(* CoDeSys 2.3 library: TcPlcUtilitiesBC.lb6 *)
(* Libraries: standard.lb6 5.6.98 11:03:02, PlcSystemBC.lb6 21.3.01 11:03:02 *)

(* Global variable list: Global_Variables *)
VAR_GLOBAL
	GLOBAL_DCF77_PULSE_SPLIT		: TIME := T#140ms;(* 0 == pulse < 140ms, 1 == pulse > 140 *)
	GLOBAL_DCF77_SEQUENCE_CHECK	: BOOL := FALSE;(* TRUE = Enable plausibility check (two telegrams are checked), FALSE = Disable check *)
END_VAR

(* Data type *)
TYPE E_ArgType :(

	ARGTYPE_UNKNOWN			:= 0,
	ARGTYPE_BYTE,
	ARGTYPE_WORD,
	ARGTYPE_DWORD,
	ARGTYPE_REAL,
	ARGTYPE_LREAL,
	ARGTYPE_SINT,
	ARGTYPE_INT,
	ARGTYPE_DINT,
	ARGTYPE_USINT,
	ARGTYPE_UINT,
	ARGTYPE_UDINT,
	ARGTYPE_STRING,
	ARGTYPE_TIME
);
END_TYPE

(* Data type *)
TYPE E_TimeZoneID :
(
	eTimeZoneID_Invalid 	:= -1,
	eTimeZoneID_Unknown  	:= 0,
	eTimeZoneID_Standard	:= 1,(* Winterzeit *)
	eTimeZoneID_Daylight 	:= 2(* Sommerzeit *)
);
END_TYPE

(* Data type *)
TYPE OTSTRUCT:
STRUCT
	wWeek:			WORD;
 	wDay:			WORD;
 	wHour:			WORD;
 	wMinute:			WORD;
 	wSecond:		WORD;
 	wMilliseconds:	WORD;
END_STRUCT
END_TYPE

(* Data type *)
TYPE T_Arg :
STRUCT
	eType				: E_ArgType			:= ARGTYPE_UNKNOWN;	(* Argument data type *)
	cbLen				: UDINT 				:= 0;							(* Argument data byte length *)
	pData				: UDINT 				:= 0;							(* Pointer to argument data *)
END_STRUCT
END_TYPE

(* Data type *)
TYPE TIMESTRUCT
STRUCT
	wYear			: WORD;
     	wMonth			: WORD;
     	wDayOfWeek		: WORD;
     	wDay			: WORD;
     	wHour			: WORD;
     	wMinute			: WORD;
     	wSecond		: WORD;
     	wMilliseconds 	: WORD;
END_STRUCT
END_TYPE

(* POU CLEARBIT32, ST *)
FUNCTION CLEARBIT32 : DWORD
VAR_INPUT
	inVal32	:	DWORD;
	bitNo	:	SINT;
END_VAR
VAR
	dwConst : DWORD := 1;
END_VAR
CLEARBIT32 := inVal32 AND NOT (SHL(dwConst,bitNo MOD 32));
END_FUNCTION

(* POU CSETBIT32, ST *)
FUNCTION CSETBIT32 : DWORD	(* conditional set bit in dword *)
VAR_INPUT
	inVal32	:	DWORD;
	bitNo	:	SINT;
	bitVal	:	BOOL;		(* value to which the bit should be set *)
END_VAR
VAR
	dwConst : DWORD := 1;
END_VAR
IF bitVal
THEN
	CSETBIT32 := inVal32 OR SHL(dwConst,bitNo MOD 32);
ELSE
	CSETBIT32 := inVal32 AND NOT (SHL(dwConst,bitNo MOD 32));
END_IF;
END_FUNCTION

(* POU DCF77_TIME, ST *)
FUNCTION_BLOCK DCF77_TIME
(* DCF77 decoder function block *)
VAR_INPUT
	DCF_PULSE	:BOOL; (* DCF77 pulse: 101010101... *)
	RUN		:BOOL; (* Enable/disable function block execution. *)
END_VAR
VAR_OUTPUT
	BUSY		:BOOL;(* TRUE = Decoding in progress *)
	ERR		:BOOL;(* Error flag: TRUE = Error, FALSE = No error *)
	ERRID		:UDINT;(* Error code *)
	ERRCNT	:UDINT;(* Error counter *)
	READY		:BOOL;  (* TRUE => CDT is valid, FALSE => CDT is not valid *)
	CDT		:DATE_AND_TIME;(* date and time information *)
END_VAR
(* 	Error codes:
	0x100	:Timeout error (no DCF-Signal)
	0x200	:Parity error
	0x300	:Wrong time or date values (e.g. Month=13)
	0x400	:Data cycle to long
	0x500	:Data cycle to short 
*)
VAR
	DataBits		: ARRAY[0..60] OF BOOL;
	BitNo		: BYTE;
	dtCurr		: DATE_AND_TIME;
	dtNext		: DATE_AND_TIME;
	tziCurr		: E_TimeZoneID;(* Time zone information extracted from latest telegram *)
	tziPrev		: E_TimeZoneID;(* Time zone information extracted from previous telegram *)
	tDiff			: TIME;(* Two telegram time difference *)
	bCheck		: BOOL := FALSE;
{library private}

	Step		: BYTE;
	StartEdge	: R_TRIG;

	RisingPulse	: R_TRIG;
	FallingPulse	: F_TRIG;
	LongPulse	: TON;
	ShortPulse	: TON;
	DetectSync	: TOF;
	NoDCFSignal	: TON;
	DCFCycleLen	: TON;

	bIsRising	: BOOL;
	bIsFalling	: BOOL;
	bIsLong		: BOOL;
	bIsShort		: BOOL;
	Working		: BOOL;

	DataValid	: BOOL;
	ParitySum1	: BYTE;
	ParitySum2	: BYTE;
	ParitySum3	: BYTE;

	i			: BYTE;
	DummyByte	: BYTE;
	DummyString	: STRING;

	Hour		: BYTE;
	Minute		: BYTE;
	Year		: BYTE;
	Month		: BYTE;
	Day			: BYTE;
{library public}
END_VAR
StartEdge( CLK := RUN );
IF  StartEdge.Q THEN
	bCheck			:= FALSE;
	BUSY			:= TRUE;
	ERR			:= FALSE;
	ERRID			:= 0;
	ERRCNT		:= 0;
	DataValid		:= FALSE;
	Working 			:= FALSE;
	BitNo			:= 0;
	NoDCFSignal( IN := FALSE );
	DCFCycleLen( IN := FALSE );
	DetectSync( IN := TRUE );
	RisingPulse( CLK := FALSE );
	FallingPulse( CLK := FALSE );
	Step			:= 10;	(* start decoding, wait for sync *)
ELSIF NOT RUN THEN
	BUSY			:= FALSE;
END_IF


IF BUSY THEN

	READY			:=FALSE;(*Ready=true is set only for one cycle*)

	RisingPulse( CLK:=DCF_PULSE ); (* detect rising edge *)
	bIsRising := RisingPulse.Q;
	FallingPulse( CLK:=DCF_PULSE );	(* detect falling edge *)
	bIsFalling := FallingPulse.Q;
	LongPulse( IN := DCF_PULSE, PT := GLOBAL_DCF77_PULSE_SPLIT );(* configurable split point *)
	IF LongPulse.Q THEN
		bIsLong := TRUE;
	END_IF
	ShortPulse( IN := DCF_PULSE, PT := T#30ms );
	IF ShortPulse.Q THEN
		bIsShort := TRUE;
	END_IF

	DetectSync( IN := DCF_PULSE, PT := T#1s500ms );(*detect the sync second*)
	IF NOT DetectSync.Q THEN
		BitNo 		:= 0;
		Step 		:= 20; (* wait for high *)
	END_IF


	NoDCFSignal( IN := DetectSync.Q, PT := T#2m );
	IF NoDCFSignal.Q THEN
		NoDCFSignal( IN := FALSE );
		ERRID		:=16#100;
		Step		:= 100;
	END_IF

	(*checking if the data cycle was longer as needed*)
	DCFCycleLen( IN:= Working , PT:=T#59s );
	IF DCFCycleLen.Q THEN
		DCFCycleLen( IN := FALSE );
		ERRID		:= 16#400;
		Step 		:= 100;
	END_IF

	CASE Step OF
		10:	(* start decoding, wait for sync *)
			BitNo := 0;

		20: (* wait for rising edge *)
			IF bIsRising THEN
				IF DataValid THEN
					DataValid 	:= FALSE;
					ERR 		:= FALSE;
					ERRID 		:= 0;
					ERRCNT 	:= 0;
					READY 		:= TRUE;
				END_IF

				IF BitNo = 0 THEN
					Working 	:= TRUE; (* set flag *)
				END_IF
				bIsLong 	:= FALSE;
				bIsShort 	:= FALSE;
				Step 		:= 30;  (* wait for falling edge *)
			END_IF

		30:	(* wait for falling pulses *)
			IF bIsFalling THEN
				IF bIsLong THEN (* long pulse *)
					DataBits[BitNo] := TRUE;
					BitNo:=BitNo+1;
				ELSIF bIsShort THEN (* short pulse *)
					DataBits[BitNo] := FALSE;
					BitNo:=BitNo+1;
				END_IF

				bIsShort := FALSE;
				bIsLong := FALSE;

				IF BitNo < 59 THEN
					Step := 20;	(* repeat *)
				ELSIF BitNo = 59 THEN
					(********************************************************************************************************)
					(*check the parity Bits....*)
					ParitySum1:=0;
					ParitySum2:=0;
					ParitySum3:=0;
					FOR i:=21 TO 28 DO (*add parity bits*)
						IF DataBits[i] THEN
							ParitySum1:=ParitySum1+1;
						END_IF
					END_FOR
					FOR i:=29 TO 35 DO
						IF DataBits[i] THEN
							ParitySum2:=ParitySum2+1;
						END_IF
					END_FOR
					FOR i:=36 TO 58 DO
						IF DataBits[i] THEN
							ParitySum3:=ParitySum3+1;
						END_IF
					END_FOR

					(*if no parity errors decode the data and set the time and date variables*)
					IF( ( ParitySum1 MOD 2 ) = 0 )
					AND ( ( ParitySum2 MOD 2 ) = 0 )
					AND ( ( ParitySum3 MOD 2 ) = 0 )
					AND ( DataBits[20] = 1 )
					AND ( DataBits[0] = 0 )
					THEN

						DummyByte:=0;
						FOR i:=21 TO 27 DO
							IF DataBits[ i ] THEN
								DummyByte := DummyByte OR SHL(BYTE#1, i - 21 );
							END_IF
						END_FOR
						Minute:= ( DummyByte AND 2#00001111 ) + ( SHR( DummyByte, 4 ) * 10 );

						DummyByte:=0;
						FOR i:=29 TO 34 DO
							IF DataBits[ i ] THEN
								DummyByte := DummyByte OR SHL(BYTE#1, i - 29 );
							END_IF
						END_FOR
						Hour:= ( DummyByte AND 2#00001111 ) + ( SHR( DummyByte, 4 ) * 10 );

						DummyByte:=0;
						FOR i:=36 TO 41 DO
							IF DataBits[ i ] THEN
								DummyByte := DummyByte OR SHL(BYTE#1, i - 36 );
							END_IF
						END_FOR
						Day := ( DummyByte AND 2#00001111 ) + ( SHR( DummyByte, 4 ) * 10 );

						DummyByte:=0;
						FOR i:=45 TO 49 DO
							IF DataBits[ i ] THEN
								DummyByte := DummyByte OR SHL(BYTE#1, i - 45 );
							END_IF
						END_FOR
						Month := ( DummyByte AND 2#00001111 ) + ( SHR( DummyByte, 4 ) * 10 );

						DummyByte:=0;
						FOR i:=50 TO 57 DO
							IF DataBits[ i ] THEN
								DummyByte := DummyByte OR SHL(BYTE#1, i - 50 );
							END_IF
						END_FOR
						Year := ( DummyByte AND 2#00001111 ) + ( SHR( DummyByte, 4 ) * 10 );

						(*Create date and time strings*)
						(*Year 2000 problem...*)
						DummyString:='DT#2';
						IF Year < 100 THEN
							DummyString:=CONCAT( DummyString, '0'  );
						END_IF
						IF Year < 10 THEN
							DummyString:=CONCAT( DummyString, '0'  );
						END_IF

						DummyString:=CONCAT( DummyString, BYTE_TO_STRING( Year ) );
						DummyString:=CONCAT( DummyString, '-'  );
						DummyString:=CONCAT( DummyString, BYTE_TO_STRING( Month ) );
						DummyString:=CONCAT( DummyString, '-' );
						DummyString:=CONCAT( DummyString, BYTE_TO_STRING( Day ) );
						DummyString:=CONCAT( DummyString, '-' );
						DummyString:=CONCAT( DummyString, BYTE_TO_STRING( Hour ) );
						DummyString:=CONCAT( DummyString, ':'  );
						DummyString:=CONCAT( DummyString, BYTE_TO_STRING( Minute ) );
						DummyString:=CONCAT( DummyString, ':00' );

						IF ( Minute > 59 ) OR ( Hour > 23 ) OR ( Day > 31 ) OR ( Day = 0 ) OR ( Month > 12 ) OR ( Month = 0 ) THEN
							ERRID		:= 16#300; (*invalid Values*)
							Step		:= 100;
						ELSE
							(*checking if the data cycle was shorter as needed*)
							IF ( DCFCycleLen.ET <T#58s ) THEN
								ERRID		:= 16#500;
								Step		:= 100;
							ELSE

								IF NOT ( DataBits[17] XOR DataBits[18] ) THEN(* bit17 = 0 and bit18 = 1 => MEZ (Standard, Winterzeit), bit17 = 1 and bit 18 = 0 => MESZ (Daylight, Sommerzeit) *)
									ERRID	:= 16#300; (*invalid MEZ/MESZ bit values*)
									Step	:= 100;
								ELSE

									dtCurr := STRING_TO_DT(DummyString);(* convert string to next time *)
	
									IF NOT GLOBAL_DCF77_SEQUENCE_CHECK THEN(* Old code: no telegram check *)
	
										DataValid	:= TRUE;
										Working		:= FALSE;
										CDT		:= dtCurr;
										BitNo 		:= 0;
										Step		:= 10;
	
									ELSE(* New code: check two telegrams *)

										IF bCheck THEN(* check the prev and current telegram*)
											tDiff := SEL( dtCurr > dtNext, dtNext - dtCurr, dtCurr - dtNext );
											tziCurr := SEL( DataBits[17], eTimeZoneID_Standard, eTimeZoneID_Daylight );

											IF ( dtNext = dtCurr )
											OR ( ( tDiff = T#1h )  AND ( tziCurr <> tziPrev ) AND DataBits[16] )(* MEZ->MESZ or MESZ->MEZ change *)
											THEN(* Time is OK *)
												bCheck 	:= TRUE;

												DataValid	:= TRUE;
												Working		:= FALSE;
												CDT		:= dtCurr;
												BitNo 		:= 0;
												Step		:= 10;
	
											ELSE(* Error  *)
												bCheck 	:= FALSE;
												ERRID	:= 16#300; (*invalid Values*)
												Step	:= 100;
											END_IF

										ELSE(* First telegram received: No telegram to check, repeat reading *)
											bCheck 	:= TRUE;
											Working	:= FALSE;
											BitNo 	:= 0;
											Step 	:= 10;
										END_IF

										dtNext := dtCurr + T#1m;(* Supposed next time *)
										tziPrev := tziCurr;(* Save this to recognize the MEZ<->MESZ time change *)
									END_IF

								END_IF

							END_IF

						END_IF

					ELSE
						ERRID		:= 16#200;(*Parity error*)
						Step		:= 100;
					END_IF

				ELSE (* > 59 *)
					BitNo 	:= 0;
					Step 	:= 10;
				END_IF
			END_IF

		100:
			bCheck	:= FALSE;
			bIsLong	:= FALSE;
			bIsShort 	:= FALSE;
			Working	:= FALSE;
			DataValid	:= FALSE;
			NoDCFSignal( IN := FALSE );
			DCFCycleLen( IN := FALSE );
			DetectSync( IN := TRUE );
			RisingPulse( CLK := FALSE );
			FallingPulse( CLK := FALSE );
			ERR 		:= TRUE;
			ERRCNT 	:= ERRCNT + 1;
			BitNo		:= 0;
			Step		:= 10;
	ELSE
		;
	END_CASE
END_IF
END_FUNCTION_BLOCK

(* POU DRAND, ST *)
FUNCTION_BLOCK DRAND
VAR_INPUT
	Seed			:	INT;
END_VAR
VAR_OUTPUT
	Num				:	REAL;
END_VAR
VAR
	R250_bInit		:	BOOL := FALSE;
	R250_Buffer		:	ARRAY[0..249] OF WORD;
	R250_Index		:	WORD;
	j,k					:	WORD;
	msb 				:	WORD := 16#8000;
	mask 				:	WORD := 16#FFFF;
	nHoldRand		:	DWORD;
	tmpRand 			: 	WORD := 0;
END_VAR
IF NOT R250_bInit THEN
	nHoldRand := Seed;
	R250_Index := 0;


	FOR j:=0 TO 249 DO
		nHoldRand := SHR( nHoldRand * 214013 + 2531011, 16) AND 16#7FFF;
		R250_Buffer[j] := DWORD_TO_WORD(nHoldRand);
	END_FOR


	FOR j:=0 TO 249 DO
		nHoldRand := SHR( nHoldRand * 214013 + 2531011, 16) AND 16#7FFF;
		IF ( nHoldRand > 16384) THEN
			R250_Buffer[j] := R250_Buffer[j] OR msb;
		END_IF
	END_FOR


	FOR j:=0 TO 15 DO
		k := 11 * j + 3;
		R250_Buffer[k] := R250_Buffer[k] AND mask;
		R250_Buffer[k] := R250_Buffer[k] OR msb;
		mask := SHR(mask, 1);
		msb  := SHR(msb, 1);
	END_FOR

	R250_bInit := TRUE;
END_IF


IF (R250_Index >= 147) THEN
	j := R250_Index - 147;
ELSE
	j := R250_Index + 103;
END_IF


tmpRand := R250_Buffer[R250_Index] XOR R250_Buffer[j];(*generate new random number*)
R250_Buffer[R250_Index] := tmpRand;



IF (R250_Index >= 249)THEN
	R250_Index := 0;
ELSE
	R250_Index := R250_Index + 1;
END_IF

Num := WORD_TO_REAL(tmpRand) / 65535;
END_FUNCTION_BLOCK

(* POU DT_TO_SYSTEMTIME, ST *)
FUNCTION DT_TO_SYSTEMTIME : TIMESTRUCT
VAR_INPUT
	DTIN		  : DATE_AND_TIME;
END_VAR
(* Day of week
	Sunday		= 0
	Monday 		= 1
	Tuesday 	= 2
	.................................
	.................................
*)
VAR
	sDT			: STRING(24);
	sYear 		: STRING(5);
	sMonth 		: STRING(3);
	sDay 		: STRING(3);
	sHour		: STRING(3);
	sMin 		: STRING(3);
	sSek 		: STRING(3);

	nDay		: BYTE;
	TS 			: TIMESTRUCT;
END_VAR
	sDT := DT_TO_STRING(DTIN);
	sYear := MID(sDT,4,4);
	sMonth := MID(sDT,2,9);
	sDay := MID(sDT,2,12);
	sHour := MID(sDT,2,15);
	sMin := MID(sDT,2,18);
	sSek := MID(sDT,2,21);
	TS.wYear := STRING_TO_WORD(sYear);
	TS.wMonth:= STRING_TO_WORD(sMonth);
	TS.wDay := STRING_TO_WORD(sDay);
	TS.wHour := STRING_TO_WORD(sHour);
	TS.wMinute := STRING_TO_WORD(sMin);
	TS.wSecond := STRING_TO_WORD(sSek);
	TS.wMilliseconds := 0;

	(*calculate the day of week*)
	nDay := DWORD_TO_BYTE( ( ( DT_TO_DWORD( DTIN ) / 86400 ) + 4 ) MOD 7 );
	TS.wDayOfWeek := nDay;

	DT_TO_SYSTEMTIME := TS;
END_FUNCTION

(* POU F_GetVersionTcPlcUtilitiesBC, ST *)
FUNCTION F_GetVersionTcPlcUtilitiesBC : UINT
VAR_INPUT
    nVersionElement       :       INT;
END_VAR
VAR
END_VAR
(* Version history:
Date          		| Version    		| created under      		| Author          	| Remark 
--------------------------------------------------------------------------------------------------------------------------------------------------------------------------------------------------------- 
Modifications:
	-----------------------------------------------------------------------
	Version: 001 (CC) Created 2001.07.24 , Compiler:2.7.501
	-Converting  functions added:
		OTSTRUCT_TO_TIME
		TIME_TO_OTSTRUCT

	Version: 002 (CC) Created 2001.07.24 , Compiler:2.7.501
	- DRAND function block added


	Version: 003 (CC) Created 2002.07.16 , Compiler:2.7.518
	- F_SwapReal function added

	Version: 004 Created 2003.03.10 , Compiler:2.9.TwinCAT Build 929. Saved as 2.7
	- DT_TO_SYSTEMTIME bug fixed. wDayOfWeek returns now  0 for Sunday and 1 for Monday an so on...

	Version: 005 Created 2003.10.24 , Compiler:2.9.TwinCAT Build 947. Saved as 2.7
	- IsFinite function and FB_BasicPID function block added
--------------------------------------------------------------------------------------------------------------------------------------------------------------------------------------------------------------------
13/05/2005    	| 1.0.6      		| V2.10.0 (Build 1230) saved as 2.7 lib	| ChristophC		| DCF77_TIME bug fixed. Array bounds exceedance corrected. F_GetVersionTcPlcUtilitiesBC added
11.02.2010	| 1.0.7			| TCAT2.11 B1540                				| ChristophC   		| DCF77_TIME short/long impuls split time changed from 110ms to 140ms. Configurable via GLOBAL_DCF77_PULSE_SPLIT variable. Telegram plausibility check.

*) 
CASE nVersionElement OF
1: (* major number *) 
       F_GetVersionTcPlcUtilitiesBC := 1;
2: (* minor number *)
       F_GetVersionTcPlcUtilitiesBC := 0;
3: (* revision number *)
       F_GetVersionTcPlcUtilitiesBC := 7;
ELSE 
   F_GetVersionTcPlcUtilitiesBC := 16#FFFF;
END_CASE
END_FUNCTION

(* POU F_REAL, ST *)
FUNCTION F_REAL : T_Arg
VAR_IN_OUT
	in		: REAL;
END_VAR
VAR
END_VAR
F_REAL.eType := ARGTYPE_REAL;
F_REAL.cbLen := SIZEOF( in );
F_REAL.pData := ADR( in );
END_FUNCTION

(* POU F_SwapReal, ST *)
FUNCTION F_SwapReal : REAL
(* Swaps Hi and Lo words of REAL variable. Do not perform any mathematical operations on swapped REAL values! *)
VAR_INPUT
	fVal		: REAL;
END_VAR
VAR
	pReal		: POINTER TO ARRAY[0..1] OF WORD;
	pResult	: POINTER TO ARRAY[0..1] OF WORD;
END_VAR
pReal := 	ADR( fVal );
pResult := ADR( F_SwapReal );

pResult^[ 0 ] := pReal^[ 1 ];
pResult^[ 1 ] := pReal^[ 0 ];
END_FUNCTION

(* POU FB_BasicPID, ST *)
FUNCTION_BLOCK FB_BasicPID
VAR_INPUT
	(* controller input  *)
	fSetpointValue		: REAL;			(* setpoint value									*)
	fActualValue		: REAL;			(* actual value										*)
	(* reset flag *)
	bReset			: BOOL;
	(* controller values *)
	fCtrlCycleTime	: REAL;			(* controller cycle time in seconds [s]			*)

	(*                                           1               Tv * s												*)
	(*	G(s) = Kp * ( 1 + ------------ + --------------- )												*)
	(*                                       Tn * s       1 + Td * s												*)

	fKp					: REAL;			(* proportional gain Kp (P)						*)
	fTn					: REAL;			(* integral gain Tn (I) [s]							*)
	fTv					: REAL;			(* derivative gain Tv (D-T1) [s]						*)
	fTd					: REAL;			(* derivative damping time Td (D-T1) [s]			*)
END_VAR
VAR_OUTPUT
	fCtrlOutput			: REAL;			(* controller output command						*)
	nErrorStatus		: UINT;				(* controller error output (0: no error; >0:error)	*)
END_VAR
VAR CONSTANT
	nERR_NOERROR			: UINT := 0;	(* no error									*)
	nERR_INVALIDPARAM		: UINT := 1;	(* invalid parameter						*)
	nERR_INVALIDCYCLETIME	: UINT := 2;	(* invalid cycle time						*)
END_VAR
VAR
	(* STATIC VARIABLE *)
	(* Internal Variable *)
	fE				: REAL := 0.0;		(* error input											*)
	fE_1			: REAL := 0.0;		(* error input z^(-1)									*)
	fY				: REAL := 0.0;		(* control output										*)
	fY_1			: REAL := 0.0;		(* control output  z^(-1)								*)
	fYP				: REAL := 0.0;		(* P-part												*)
	fYI				: REAL := 0.0;		(* I-part												*)
	fYI_1			: REAL := 0.0;		(* I-part  z^(-1)											*)
	fYD				: REAL := 0.0;		(* D-T1-part											*)
	fYD_1			: REAL := 0.0;		(* D-T1-part  z^(-1)										*)
	(* Internal Parameter *)
	bInit			: BOOL	:= TRUE;	(* initialization flag for first cycle						*)
	bIsIPart		: BOOL	:= FALSE;	(* I-part active ?										*)
	bIsDPart		: BOOL	:= FALSE;	(* D-part active ?										*)

	fDi				: REAL	:= 0.0;		(* internal I param										*)
	fDd				: REAL	:= 0.0;		(* internal D param									*)
	fCd				: REAL	:= 0.0;		(* internal D param									*)

	fCtrlCycleTimeOld	: REAL	:= 0.0;
	fKpOld				: REAL	:= 0.0;
	fTnOld				: REAL	:= 0.0;
	fTvOld				: REAL	:= 0.0;
	fTdOld				: REAL	:= 0.0;
END_VAR
(* init necessary? *)
IF (fCtrlCycleTime <> fCtrlCycleTimeOld) OR (fKp <> fKpOld) OR (fTn <> fTnOld) OR (fTv <> fTvOld) OR (fTd <> fTdOld)
THEN
	bInit := TRUE;
END_IF

(* controller init *)
IF bInit OR bReset
THEN
	(* reset internal and external variables *)
	fE	:= fE_1			:= 0.0;
	fY	:= fY_1			:= 0.0;
	fYP	:= 0.0;
	fYI	:= fYI_1		:= 0.0;
	fYD	:= fYD_1		:= 0.0;
	fCtrlOutput			:= 0.0;
	bIsIPart			:= FALSE;
	bIsDPart			:= FALSE;
	fCtrlOutput			:= 0.0;
	nErrorStatus		:= nERR_NOERROR;

	(* check cycle time parameter: (CycleTime > 0 AND CycleTme <= 60) *)
	IF ( fCtrlCycleTime <= 0)
	THEN
		nErrorStatus := nERR_INVALIDCYCLETIME;
		RETURN;
	END_IF;

	(* check controller parameters: (Tn, Tv, Td >= 0) *)
	IF ( (fTn < 0) OR (fTv < 0) OR (fTd < fCtrlCycleTime/2.0) ) THEN
		nErrorStatus := nERR_INVALIDPARAM;
		RETURN;
	END_IF;

	(* I-part *)
	IF( fTn > 0.0 ) THEN
		fDi := (fKp * fCtrlCycleTime) / (2.0 * fTn);
		bIsIPart := TRUE;
	ELSE
		fDi := 0.0;
		bIsIPart := FALSE;
	END_IF;

	(* D-part *)
	IF( fTv > 0.0 ) AND (fTd > 0.0)
         THEN
		fDd := (fKp * fTv) / (fTd + fCtrlCycleTime / 2.0);
		fCd := (fTd - fCtrlCycleTime / 2.0) / (fTd + fCtrlCycleTime / 2.0);
		bIsDPart := TRUE;
	ELSE
		fDd := 0.0;
		fCd := 0.0;
		bIsDPart := FALSE;
	END_IF;

	(* reset *)
	IF bReset
	THEN
		RETURN;
	END_IF


	(* set internal init flag *)
	fCtrlCycleTimeOld 	:= fCtrlCycleTime;
	fKpOld 				:= fKp;
	fTnOld 					:= fTn;
	fTvOld 					:= fTv;
	fTdOld 					:= fTd;
	bInit					:= FALSE;
END_IF;



(* 3. save old variable *)
fE_1	:= fE;
fY_1	:= fY;
fYI_1	:= fYI;
fYD_1	:= fYD;

(* 4. set error/deviation input *)
fE	:= fSetpointValue - fActualValue;

(* 5. YP-part *)
fYp		:= fKp * fE;

(* 6. YI-part *)
IF bIsIPart THEN
	fYI := fYI_1 + fDi * (fE + fE_1);					(* normal I-part calculation *)
ELSE
	fYI			:= 0.0;
END_IF;

(* 7. YD-part *)
IF bIsDPart THEN
	fYD	:=  fCd * fYD_1 + fDd * (fE - fE_1);
ELSE
	fYD	:= 0.0;
END_IF;

(* 8. Ysum = YP + YI + YD *)
fY	:= fYP + fYI + fYD;

(* 10. set controller output *)
fCtrlOutput := fY;
END_FUNCTION_BLOCK

(* POU GETBIT32, ST *)
FUNCTION GETBIT32 : BOOL
VAR_INPUT
	inVal32	:	DWORD;
	bitNo	:	SINT;
END_VAR
VAR
	dwConst : DWORD := 1;
END_VAR
IF ( inVal32 AND SHL( dwConst,bitNo MOD 32 ) ) > 0
THEN
	GETBIT32 := TRUE;
ELSE
	GETBIT32 := FALSE;
END_IF;
END_FUNCTION

(* POU IsFinite, ST *)
FUNCTION IsFinite : BOOL
(*	Function returns a nonzero value (TRUE) if its argument x is not infinite, that is, if INF < x < +INF. It returns 0 (FALSE) if the argument is infinite or a NaN *)
VAR_INPUT
	x				:T_ARG;
END_VAR
VAR
	ptrDouble		: POINTER TO ARRAY[ 0..1] OF  DWORD;
	ptrSingle			: POINTER TO  DWORD;
END_VAR
(*
	Double precision (LREAL )
	If exponent=2047 and fraction is nonzero, then x = Nan ("Not a number") 
	If exponent=2047 and fraction is zero and sign is 1, then x = "-Infinity" 
	If exponent=2047 and fraction is zero and sign is 0, then x = "Infinity"

	Single precision (REAL):
	If exponent=255 and fraction is nonzero, then x = Nan ("Not a number") 
	If exponent=255 and fraction is zero and sign is 1, then x = "-Infinity" 
	If exponent=255 and fraction is zero and sign is 0, then x = "Infinity"
*)
IF x.eType = ARGTYPE_LREAL THEN
	ptrDouble := x.pData;

	IF ( ptrDouble^[ 1 ] AND 16#7FF0_0000 )  = 16#7FF0_0000 THEN (*exponent  = 2047*)
		IF ( ( ptrDouble^[ 1 ] AND 16#000F_FFFF ) OR ( ptrDouble^[ 0 ] ) ) = 0 THEN (*fraction = 0*)
			IF ( ptrDouble^[ 1 ] AND 16#8000_0000 ) =  0 THEN (* sign = 0*)
				IsFinite := FALSE; (*+Infinity*)
			ELSE (* sign = 1*)
				IsFinite := FALSE; (*-Inifinity*)
			END_IF
		ELSE (* fraction <> 0 *)
			IsFinite := FALSE; (*NaN*)
		END_IF
	ELSE
		IsFinite := TRUE;
	END_IF

ELSIF x.eType = ARGTYPE_REAL THEN
	ptrSingle := x.pData;

	IF ( ptrSingle^ AND 16#0000_7F80 )  = 16#0000_7F80 THEN (*exponent  = 255*)

		IF ( ptrSingle^ AND 16#FFFF_007F ) = 0 THEN (*fraction bits = 0*)

			IF ( ptrSingle^ AND 16#0000_8000 ) =  0 THEN (* sign bit = 0*)
				IsFinite := FALSE; (*+Infinity*)
			ELSE (* sign = 1*)
				IsFinite := FALSE; (*-Inifinity*)
			END_IF
		ELSE (* fraction bits <> 0 *)
			IsFinite := FALSE; (*NaN*)
		END_IF
	ELSE
		IsFinite := TRUE;
	END_IF
END_IF
END_FUNCTION

(* POU OTSTRUCT_TO_TIME, ST *)
FUNCTION OTSTRUCT_TO_TIME : TIME
VAR_INPUT
	OTIN	:OTSTRUCT;
END_VAR
VAR
	tmpMilli: 	DWORD;
END_VAR
tmpMilli := 	WORD_TO_DWORD(OTIN.wMilliseconds) +
		  	( WORD_TO_DWORD(OTIN.wSecond) * 1000 ) +
			( WORD_TO_DWORD(OTIN.wMinute) * 60000 ) +
			( WORD_TO_DWORD(OTIN.wHour) * 3600000 ) +
			( WORD_TO_DWORD(OTIN.wDay) * 86400000 ) +
			( WORD_TO_DWORD(OTIN.wWeek) *604800000 );

OTSTRUCT_TO_TIME := DWORD_TO_TIME( tmpMilli );
END_FUNCTION

(* POU ReadWriteTerminalReg, ST *)
FUNCTION_BLOCK ReadWriteTerminalReg
VAR_INPUT
	STATE				:BYTE;		(*Terminal Status Byte*)
	DATAIN				:WORD;		(*Terminal Data IN*)
	REGNO				:BYTE;
	READ				:BOOL;
	WRITE				:BOOL;
	TMOUT				:TIME;
	NEWREGVALUE		:WORD;
END_VAR
VAR_OUTPUT
	CTRL				:BYTE;		(*Terminal Control Byte*)
	DATAOUT			:WORD;		(*Terminal Data OUT*)
	BUSY				:BOOL;
	ERR				:BOOL;
	ERRID				:UDINT;
	CURREGVALUE		:WORD;
	(*
		Error codes:
		0			=No error;
		0x100		=Timeout error
		0x200		= Parameter error
		0x300		= Writing not successfully ( writing to the register not allowed )
	*)
END_VAR
VAR
	STEP				:BYTE	:= 	16#0;
	ErrStep 				:BYTE	:=	0;
(*
		if Timeout and
		ErrStep = 0x20		=> 	( disabling the write protection )
		ErrStep = 0x30		=>	( during write request )
		ErrStep = 0x40		=>	( enabling  the write protection )
		ErrStep = 0x60		=>	( during read request )

*)
	RisingEdge_Read	:R_TRIG;
	RisingEdge_Write		:R_TRIG;
	TimerTON			:TON;
	bCheckSuccess		:BOOL	:= FALSE;
END_VAR
RisingEdge_Read(CLK:=READ);
RisingEdge_Write(CLK:= WRITE);


IF ( RisingEdge_Read.Q XOR RisingEdge_Write.Q )  THEN
	bCheckSuccess := FALSE;
	ErrStep 	:= 0;
	CURREGVALUE:=0;
	CTRL:=0;

	IF REGNO < 64 THEN
		BUSY:=TRUE;
		ERR:=FALSE;
		ERRID:=0;
		Step:=16#1;
	ELSE
		BUSY := FALSE;
		ERR:=TRUE;
		ERRID:=16#200;
		Step := 16#0;
	END_IF

END_IF


CASE Step OF
	16#0:
		(*do nothing*);
	16#1:
		IF READ THEN
			bCheckSuccess := FALSE;
			Step := 16#50;
		ELSE	 (*write*)
			bCheckSuccess := TRUE;
			Step := 16#10;
		END_IF

	(***************			WRITE the Terminal Register			**************************)
	16#10:
		CTRL:=2#11000000;
		CTRL:=CTRL OR 16#1F ;				(*Select Register 31*)
		DATAOUT:=16#1235;					(*Write Protection OFF*)
		Step := 16#20;
	16#20:
		IF ( STATE=16#9F ) THEN
			CTRL:=2#11000000;
			CTRL:=Ctrl OR REGNO ;
			DATAOUT:=NEWREGVALUE;		(*Set new Value*)
			Step := 16#30;
		END_IF
	16#30:
		IF ( CTRL=(STATE OR 2#01000000) ) THEN
			CTRL:=2#11000000;
			CTRL:=CTRL OR 16#1F ;			(*Select Register 31*)
			DATAOUT:=0;					(*Write protection ON*)
			Step := 16#40;
		END_IF
	16#40:
		IF ( CTRL=(STATE OR 2#01000000) ) THEN
			Step := 16#50;
		END_IF

	(***************			READ the Terminal Register			**************************)
	16#50:
		CTRL:=2#10000000;
		CTRL:=Ctrl OR REGNO;
		Step := 16#60;
	16#60:
		IF ( CTRL=STATE ) THEN
			CURREGVALUE:=DATAIN;
			Busy:=FALSE;
			CTRL:=0;
			Step:=16#0;

			IF ( bCheckSuccess AND ( NEWREGVALUE <> CURREGVALUE ) )THEN
				ERR := TRUE;
				ERRID := 16#300;
			END_IF

		END_IF

END_CASE




TimerTON( PT:=TMOUT,  IN:=BUSY  );
IF TimerTON.Q THEN
	Busy:=FALSE;
	ERR:=TRUE;
	ERRID:=16#100;
	ErrStep := Step;
	Step:=16#0;
	CTRL:=0;
	CURREGVALUE:=0;
END_IF
END_FUNCTION_BLOCK

(* POU RTC, ST *)
FUNCTION_BLOCK RTC
VAR_INPUT
	EN				:BOOL;
	PDT			:DATE_AND_TIME;
END_VAR
VAR_OUTPUT
	Q				:BOOL;
	CDT			:DATE_AND_TIME;
END_VAR
VAR
	OldTick			:DWORD:=0;
	CurrTick			:DWORD:=0;
	nMilliDiff			:DWORD:=0;
	nMilliRest		:DWORD:=0;
	RisingEdge		:R_TRIG;
END_VAR
CurrTick:=GetSysTick(TRUE);
(*CurrTick:=%MD4088;    changed 20001.02.08 C.C.*)
(*GetSysTick has dummy parameter:    changed 20001.03.21 C.C.*)
RisingEdge( CLK:=EN );

IF RisingEdge.Q THEN
	nMilliRest:=0;
	CDT:=PDT;
	Q:=TRUE;
ELSE
	IF OldTick > CurrTick THEN
		nMilliDiff:= ( 16#FFFFFFFF - OldTick ) + CurrTick +1 +nMilliRest;
	ELSE
		nMilliDiff:=CurrTick - OldTick + nMilliRest;
	END_IF

	nMilliRest:=nMilliDiff MOD 1000;
	CDT:= DWORD_TO_DT( DT_TO_DWORD(CDT) + ( nMilliDiff / 1000 ) );
END_IF

OldTick:=CurrTick;
END_FUNCTION_BLOCK

(* POU RTC_EX, ST *)
FUNCTION_BLOCK RTC_EX
VAR_INPUT
	EN				:BOOL;
	PDT			:DATE_AND_TIME;
	PMSEK			:DWORD;
END_VAR
VAR_OUTPUT
	Q				:BOOL;
	CDT			:DATE_AND_TIME;
	CMSEK			:DWORD;
END_VAR
VAR
	OldTick			:DWORD:=0;
	CurrTick			:DWORD:=0;
	nMilliDiff			:DWORD:=0;
	nMilliRest		:DWORD:=0;
	RisingEdge		:R_TRIG;
END_VAR
CurrTick:=GetSysTick(TRUE);
(*CurrTick:=%MD4088;    changed 20001.02.08 C.C.*)
(*GetSysTick has dummy parameter:    changed 20001.03.21 C.C.*)
RisingEdge( CLK:=EN );

IF RisingEdge.Q THEN
	nMilliRest:=PMSEK;
	CDT:=PDT;
	Q:=TRUE;
ELSE
	IF OldTick > CurrTick THEN
		nMilliDiff:= ( 16#FFFFFFFF - OldTick ) + CurrTick +1 +nMilliRest;
	ELSE
		nMilliDiff:=CurrTick - OldTick + nMilliRest;
	END_IF

	nMilliRest:=nMilliDiff MOD 1000;
	CDT:= DWORD_TO_DT( DT_TO_DWORD(CDT) + ( nMilliDiff / 1000 ) );
END_IF

OldTick:=CurrTick;
CMSEK:=nMilliRest;
END_FUNCTION_BLOCK

(* POU SETBIT32, ST *)
FUNCTION SETBIT32 : DWORD
VAR_INPUT
	inVal32	:	DWORD;
	bitNo	:	SINT;
END_VAR
VAR
	dwConst : DWORD := 1;
END_VAR
SETBIT32 := inVal32 OR SHL( dwConst,bitNo MOD 32 );
END_FUNCTION

(* POU SYSTEMTIME_TO_DT, ST *)
FUNCTION SYSTEMTIME_TO_DT : DATE_AND_TIME
VAR_INPUT
	TIMESTR			: TIMESTRUCT;
END_VAR
VAR
	TempString			: STRING;
	nSeconds			: DWORD;		
END_VAR
	TempString:='DT#';
	TempString:=CONCAT( TempString, WORD_TO_STRING( TIMESTR.wYear ) );
	TempString:=CONCAT( TempString, '-'  );
	TempString:=CONCAT( TempString, WORD_TO_STRING( TIMESTR.wMonth ) );
	TempString:=CONCAT( TempString, '-' );
	TempString:=CONCAT( TempString, WORD_TO_STRING( TIMESTR.wDay ) );
	TempString:=CONCAT( TempString, '-' );
	TempString:=CONCAT( TempString, WORD_TO_STRING( TIMESTR.wHour ) );
	TempString:=CONCAT( TempString, ':'  );
	TempString:=CONCAT( TempString, WORD_TO_STRING( TIMESTR.wMinute ) );
	TempString:=CONCAT( TempString, ':' );
	TempString:=CONCAT( TempString, WORD_TO_STRING( TIMESTR.wSecond ) );

	(*Round the milliseconds to seconds*)
	nSeconds := DT_TO_DWORD( STRING_TO_DT( TempString ) );
	IF ( TIMESTR.wMilliseconds > 499 ) THEN
		nSeconds := nSeconds + 1;
	END_IF

	SYSTEMTIME_TO_DT:=DWORD_TO_DT( nSeconds);
END_FUNCTION

(* POU TIME_TO_OTSTRUCT, ST *)
FUNCTION TIME_TO_OTSTRUCT : OTSTRUCT(* Converts TIME data type to operating time struct  with weeks, days, hours, minutes, *)
VAR_INPUT
	TIN			:TIME;
END_VAR
VAR
	tmpMilli: 	DWORD;
END_VAR
	tmpMilli:=TIME_TO_DWORD(TIN);

	TIME_TO_OTSTRUCT.wMilliseconds :=DWORD_TO_WORD( tmpMilli MOD 1000 );
	(* 1000 *)
	TIME_TO_OTSTRUCT.wSecond :=DWORD_TO_WORD ( ( tmpMilli / 1000 ) MOD 60 );
	(* 1000*60 *)
	TIME_TO_OTSTRUCT.wMinute := DWORD_TO_WORD( ( tmpMilli / 60000 ) MOD 60 );
	(* 1000*60*60 *)
	TIME_TO_OTSTRUCT.wHour := DWORD_TO_WORD( ( tmpMilli / 3600000 ) MOD 24 );
	(*1000*60*60*24 *)
	TIME_TO_OTSTRUCT.wDay := DWORD_TO_WORD( ( tmpMilli / 86400000 ) MOD 7 );
	(* 1000*60*60*24*7 *)
	TIME_TO_OTSTRUCT.wWeek:=DWORD_TO_WORD( ( tmpMilli / 604800000 ) );
END_FUNCTION
